ABB RAPID module: Module_Tarea1.mod

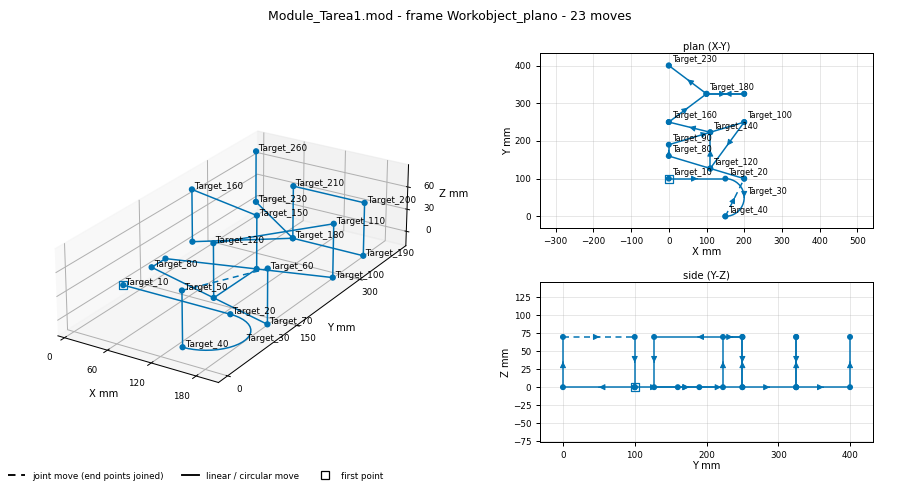
[picture p0: tool path of Module_Tarea1.mod in frame Workobject_plano, 23 of 50 moves have a stored position in this frame; points joined in program order, loops and branches not executed]
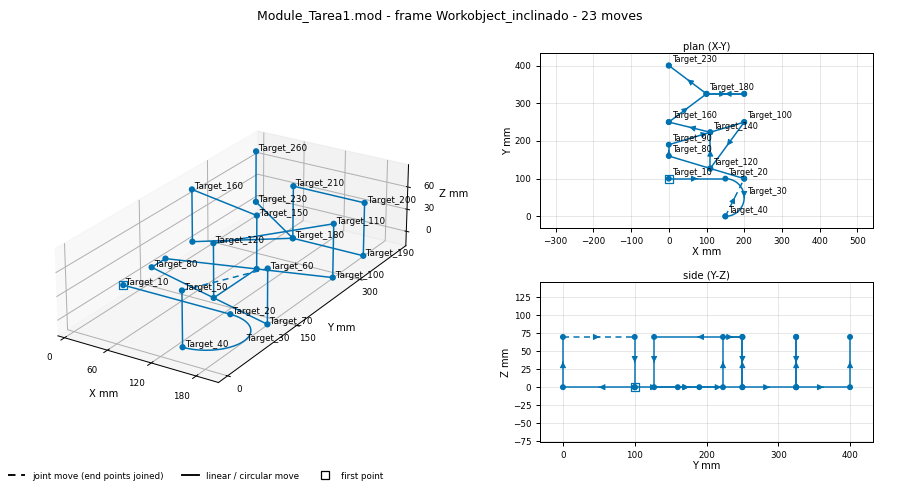
[picture p1: tool path of Module_Tarea1.mod in frame Workobject_inclinado, 23 of 50 moves have a stored position in this frame; points joined in program order, loops and branches not executed]
MODULE Module1
    CONST robtarget Target_10:=[[0,100,0],[0,1,0,0],[0,-2,1,0],[9E+09,9E+09,9E+09,9E+09,9E+09,9E+09]];
    CONST robtarget Target_20:=[[150,100,0],[0,1,0,0],[0,-2,1,0],[9E+09,9E+09,9E+09,9E+09,9E+09,9E+09]];
    CONST robtarget Target_30:=[[200,50,0],[0,1,0,0],[0,-2,1,0],[9E+09,9E+09,9E+09,9E+09,9E+09,9E+09]];
    CONST robtarget Target_40:=[[150,0,0],[0,1,0,0],[0,-2,1,0],[9E+09,9E+09,9E+09,9E+09,9E+09,9E+09]];
    CONST robtarget Target_50:=[[150,0,70],[0,1,0,0],[-1,-2,1,0],[9E+09,9E+09,9E+09,9E+09,9E+09,9E+09]];
    CONST robtarget Target_60:=[[200,100,70],[0,1,0,0],[-1,-1,0,1],[9E+09,9E+09,9E+09,9E+09,9E+09,9E+09]];
    CONST robtarget Target_70:=[[200,100,0],[0,1,0,0],[-1,-1,0,1],[9E+09,9E+09,9E+09,9E+09,9E+09,9E+09]];
    CONST robtarget Target_80:=[[0,160,0],[0,1,0,0],[-1,-1,0,1],[9E+09,9E+09,9E+09,9E+09,9E+09,9E+09]];
    CONST robtarget Target_90:=[[0,190,0],[0,1,0,0],[-1,-1,0,1],[9E+09,9E+09,9E+09,9E+09,9E+09,9E+09]];
    CONST robtarget Target_100:=[[200,250,0],[0,1,0,0],[-1,-1,0,1],[9E+09,9E+09,9E+09,9E+09,9E+09,9E+09]];
    CONST robtarget Target_110:=[[200,250,70],[0,1,0,0],[-1,-1,0,1],[9E+09,9E+09,9E+09,9E+09,9E+09,9E+09]];
    CONST robtarget Target_120:=[[110,127,70],[0,1,0,0],[-1,-1,0,1],[9E+09,9E+09,9E+09,9E+09,9E+09,9E+09]];
    CONST robtarget Target_130:=[[110,127,0],[0,1,0,0],[-1,-1,0,1],[9E+09,9E+09,9E+09,9E+09,9E+09,9E+09]];
    CONST robtarget Target_140:=[[110,222.972,0],[0,1,0,0],[-1,-1,0,1],[9E+09,9E+09,9E+09,9E+09,9E+09,9E+09]];
    CONST robtarget Target_150:=[[110,222.972,70],[0,1,0,0],[-1,-1,0,1],[9E+09,9E+09,9E+09,9E+09,9E+09,9E+09]];
    CONST robtarget Target_160:=[[0,250,70],[0,1,0,0],[-1,-1,0,1],[9E+09,9E+09,9E+09,9E+09,9E+09,9E+09]];
    CONST robtarget Target_170:=[[0,250,0],[0,1,0,0],[-1,-1,0,1],[9E+09,9E+09,9E+09,9E+09,9E+09,9E+09]];
    CONST robtarget Target_180:=[[100,324.945,0],[0,1,0,0],[-1,-1,0,1],[9E+09,9E+09,9E+09,9E+09,9E+09,9E+09]];
    CONST robtarget Target_190:=[[200,324.945,0],[0,1,0,0],[-1,-1,0,1],[9E+09,9E+09,9E+09,9E+09,9E+09,9E+09]];
    CONST robtarget Target_200:=[[200,324.945,70],[0,1,0,0],[-1,-1,0,1],[9E+09,9E+09,9E+09,9E+09,9E+09,9E+09]];
    CONST robtarget Target_210:=[[100,324.945,70],[0,1,0,0],[-1,-1,0,1],[9E+09,9E+09,9E+09,9E+09,9E+09,9E+09]];
    CONST robtarget Target_220:=[[100,324.945,0],[0,1,0,0],[-1,-1,0,1],[9E+09,9E+09,9E+09,9E+09,9E+09,9E+09]];
    CONST robtarget Target_230:=[[0,400,0],[0,1,0,0],[-1,-1,0,1],[9E+09,9E+09,9E+09,9E+09,9E+09,9E+09]];
    CONST robtarget Target_240:=[[500.678899716,-0.000435316,594.778188],[0.258819045,0,-0.965925826,0],[-1,-2,1,1],[9E+09,9E+09,9E+09,9E+09,9E+09,9E+09]];
    CONST robtarget Target_260:=[[0,400,70],[0,1,0,0],[-1,-1,0,1],[9E+09,9E+09,9E+09,9E+09,9E+09,9E+09]];
!***********************************************************
    !
    ! Module:  Module1
    !
    ! Description:
    !   <Insert description here>
    !
    ! Author: AndresMedina
    !
    ! Version: 1.0
    !
    !***********************************************************


    !***********************************************************
    !
    ! Procedure main
    !
    !   This is the entry point of your program
    !
    !***********************************************************
    PROC main()
        IF DI_01=1 AND DI_02=0 THEN
          path_plano;
        ELSEIF DI_01=0 AND DI_02=1 THEN
          path_inclinado;
        ENDIF
    ENDPROC
    PROC path_plano()
        MoveJ Target_240,v300,z0,Tip\WObj:=wobj0;
        MoveJ Target_10,v300,z0,Tip\WObj:=Workobject_plano;
        MoveL Target_20,v100,z1,Tip\WObj:=Workobject_plano;
        MoveC Target_30,Target_40,v100,z1,Tip\WObj:=Workobject_plano;
        MoveL Target_50,v100,z1,Tip\WObj:=Workobject_plano;
        MoveJ Target_60,v100,z1,Tip\WObj:=Workobject_plano;
        MoveL Target_70,v100,z1,Tip\WObj:=Workobject_plano;
        MoveL Target_80,v100,z1,Tip\WObj:=Workobject_plano;
        MoveL Target_90,v100,z1,Tip\WObj:=Workobject_plano;
        MoveL Target_100,v100,z1,Tip\WObj:=Workobject_plano;
        MoveL Target_110,v100,z1,Tip\WObj:=Workobject_plano;
        MoveL Target_120,v100,z1,Tip\WObj:=Workobject_plano;
        MoveL Target_130,v100,z1,Tip\WObj:=Workobject_plano;
        MoveL Target_140,v100,z1,Tip\WObj:=Workobject_plano;
        MoveL Target_150,v100,z1,Tip\WObj:=Workobject_plano;
        MoveL Target_160,v100,z1,Tip\WObj:=Workobject_plano;
        MoveL Target_170,v100,z1,Tip\WObj:=Workobject_plano;
        MoveL Target_180,v100,z1,Tip\WObj:=Workobject_plano;
        MoveL Target_190,v100,z1,Tip\WObj:=Workobject_plano;
        MoveL Target_200,v100,z1,Tip\WObj:=Workobject_plano;
        MoveL Target_210,v100,z1,Tip\WObj:=Workobject_plano;
        MoveL Target_220,v100,z1,Tip\WObj:=Workobject_plano;
        MoveL Target_230,v100,z1,Tip\WObj:=Workobject_plano;
        MoveL Target_260,v300,z0,Tip\WObj:=Workobject_plano;
        MoveJ Target_240,v300,z0,Tip\WObj:=wobj0;
    ENDPROC
    PROC path_inclinado()
        MoveJ Target_240,v300,z0,Tip\WObj:=wobj0;
        MoveJ Target_10,v300,z0,Tip\WObj:=Workobject_inclinado;
        MoveL Target_20,v100,z1,Tip\WObj:=Workobject_inclinado;
        MoveC Target_30,Target_40,v100,z1,Tip\WObj:=Workobject_inclinado;
        MoveL Target_50,v100,z1,Tip\WObj:=Workobject_inclinado;
        MoveJ Target_60,v100,z1,Tip\WObj:=Workobject_inclinado;
        MoveL Target_70,v100,z1,Tip\WObj:=Workobject_inclinado;
        MoveL Target_80,v100,z1,Tip\WObj:=Workobject_inclinado;
        MoveL Target_90,v100,z1,Tip\WObj:=Workobject_inclinado;
        MoveL Target_100,v100,z1,Tip\WObj:=Workobject_inclinado;
        MoveL Target_110,v100,z1,Tip\WObj:=Workobject_inclinado;
        MoveL Target_120,v100,z1,Tip\WObj:=Workobject_inclinado;
        MoveL Target_130,v100,z1,Tip\WObj:=Workobject_inclinado;
        MoveL Target_140,v100,z1,Tip\WObj:=Workobject_inclinado;
        MoveL Target_150,v100,z1,Tip\WObj:=Workobject_inclinado;
        MoveL Target_160,v100,z1,Tip\WObj:=Workobject_inclinado;
        MoveL Target_170,v100,z1,Tip\WObj:=Workobject_inclinado;
        MoveL Target_180,v100,z1,Tip\WObj:=Workobject_inclinado;
        MoveL Target_190,v100,z1,Tip\WObj:=Workobject_inclinado;
        MoveL Target_200,v100,z1,Tip\WObj:=Workobject_inclinado;
        MoveL Target_210,v100,z1,Tip\WObj:=Workobject_inclinado;
        MoveL Target_220,v100,z1,Tip\WObj:=Workobject_inclinado;
        MoveL Target_230,v100,z1,Tip\WObj:=Workobject_inclinado;
        MoveL Target_260,v300,z0,Tip\WObj:=Workobject_inclinado;
        MoveJ Target_240,v300,z0,Tip\WObj:=wobj0;
    ENDPROC
ENDMODULE
